FUNCTION_BLOCK CU020DialogContent EXTENDS TcoCore.TcoInputDialogContentContainer
VAR_INPUT
END_VAR
VAR_OUTPUT
END_VAR
VAR
	{attribute addProperty Name "<#Recipe#>"}
	Recipe:STRING;
	{attribute addProperty Name "<#Qantity#>"}
	RequiredQuantity:INT;
	{attribute addProperty Name "<#Timeout#>"}
	Timeout:DATE_AND_TIME;
	{attribute addProperty Name "<#Exclude#>"}
	Exclude:BOOL;

END_VAR

END_FUNCTION_BLOCK

(* stored: Version 1.1.0.1
   POU CU020DialogContent: Id {160cede1-cc1b-4968-a87a-4c89fe82eefc}, SpecialFunc None *)
